INTERFACE I_PROCESS_NEST2_4 EXTENDS I_GENERAL_OBJECT

METHOD M_EnduranceRun : BOOL
VAR_INPUT
  udiCycles:                            UDINT;
  stEnduranceRunParams:                 ST_RECIPE_ENDURANCE_RUN;
END_VAR
END_METHOD

METHOD M_LeakTest1 : BOOL
VAR_INPUT
  stLeakTest1Params:                 ST_RECIPE_LEAK_TEST1;
END_VAR
END_METHOD

METHOD M_MeasureStrokeLength : BOOL
VAR_INPUT
  bCylinderDecoupled:             BOOL;
  rWorkForceA:                    REAL;
  rWorkForceB:                    REAL;
  rLoadForceA:                    REAL;
  rLoadForceB:                    REAL;
END_VAR
END_METHOD

METHOD M_MoveToSetPos : BOOL
VAR_INPUT
END_VAR
END_METHOD

METHOD M_Reset : BOOL
VAR_INPUT
END_VAR
END_METHOD

METHOD M_ResetDistance : BOOL
VAR_INPUT
END_VAR
END_METHOD

METHOD M_SetEnableState : BOOL
VAR_INPUT
  bEnable:              BOOL;
END_VAR
END_METHOD

METHOD M_SetReady : BOOL
VAR_INPUT
END_VAR
END_METHOD

METHOD M_Stop : BOOL
END_METHOD

METHOD M_StopEngine : BOOL
VAR_INPUT
END_VAR
END_METHOD

METHOD M_VentCylinder : BOOL
VAR_INPUT
  bCylinderDecoupled:             BOOL;
  uiVentCount:                    UINT;
  rWorkForceA:                    REAL;
  rWorkForceB:                    REAL;
  rLoadForceA:                    REAL;
  rLoadForceB:                    REAL;
END_VAR
END_METHOD

PROPERTY P_CurrentCycle : UDINT
GET
END_GET
END_PROPERTY

PROPERTY P_EnableState : BOOL
GET
END_GET
END_PROPERTY

PROPERTY P_NokDifference : REAL
GET
END_GET
END_PROPERTY

PROPERTY P_NokLimitInPercent : UINT
GET
END_GET
END_PROPERTY

PROPERTY P_ReadyState : BOOL
GET
END_GET
END_PROPERTY

PROPERTY P_SerialNr : STRING
GET
END_GET
SET
END_SET
END_PROPERTY

PROPERTY P_Timer : STRING
GET
END_GET
END_PROPERTY

END_INTERFACE

(* stored: Version 1.1.0.1, ProductVersion 3.1.4024.12
   Itf I_PROCESS_NEST2_4: Id {6f696aaf-e8af-4351-8608-42dfd3bffb6c}
   Method M_EnduranceRun: Id {f617bdb5-2346-4bf3-b769-8d3e40cc76be}
   Method M_LeakTest1: Id {2adb96ae-fd5c-4ece-bb88-a9737ebaef35}
   Method M_MeasureStrokeLength: Id {ed996126-2858-4368-8d8b-e6f77fde652f}
   Method M_MoveToSetPos: Id {1e57c0b3-56ba-47b6-9c1a-137b29f7fc03}
   Method M_Reset: Id {d57b43d5-154c-4286-b50b-92504feea29a}
   Method M_ResetDistance: Id {66beff43-dad1-4d8d-93b4-dddf76b7c287}
   Method M_SetEnableState: Id {e748f508-7460-4608-bcd9-24c60df37e46}
   Method M_SetReady: Id {2fe4d089-4209-4b6e-968b-b6d8bd2a5128}
   Method M_Stop: Id {dd7d451f-ad91-4c13-bb23-9981be66abb8}
   Method M_StopEngine: Id {31c86038-9414-42fd-a997-7cfd6b89aa13}
   Method M_VentCylinder: Id {785aa2c9-964a-47eb-8dc8-ea77ef867a89}
   Property P_CurrentCycle: Id {5be5f4b9-f9aa-49d9-9c6c-c493358b6a97}
   Get Get: Id {b6a7aad0-83c7-4025-bd65-3007e3bc4182}
   Property P_EnableState: Id {5a8f3172-1a32-470f-a9e7-01d6a343eb69}
   Get Get: Id {700f6fd8-6e5d-4586-a6a4-0457e22d4347}
   Property P_NokDifference: Id {3ee0d4f6-8bb2-4809-8cb0-0b0e55290687}
   Get Get: Id {6559f1de-cae7-4ddc-9d9e-817c4609fff3}
   Property P_NokLimitInPercent: Id {eb5f006f-8c83-4461-8d15-305d1e73ffd6}
   Get Get: Id {8aa00b9a-eafb-429a-a6a0-770f86da1cc1}
   Property P_ReadyState: Id {2ad007eb-173e-41f1-8228-f61cd49a53b8}
   Get Get: Id {e59d8284-0a56-4adc-83b7-924c13874db0}
   Property P_SerialNr: Id {a78d2b4f-c30b-4d7f-ad07-1c7d34455ef3}
   Get Get: Id {558e5a12-a10e-4b0d-ad88-d117f0a6a7b1}
   Set Set: Id {ebd5d485-93f0-4e93-8512-cdb1e4a9bcf5}
   Property P_Timer: Id {cc388c17-8d09-4e1b-b6ba-f296872dd93e}
   Get Get: Id {c0306dbc-7672-4513-a910-d0b803799404} *)
